// TIA Portal V20 export
TYPE "LConSMC_typeJogDynamics"
// Tippdynamiken / Jog dynamics
// stored: Access Published
   STRUCT
      acceleration : Real := 0.2;   // Beschleunigung in Achseinheit / Acceleration value: Units are taken from the TO
      deceleration : Real := 0.2;   // Verzögerung in Achseinheit / Deceleration value: Units are taken from the TO
      jerk : Real := 0.4;   // Ruckbegrenzung in Achseinheit / Jerk value : Units are taken from the TO
   END_STRUCT;
END_TYPE
